(*

## Short summary
An interface to provide a scope selector for configurations in cycle managers.

.. <legal notes>

legal notes
=================
| SPDX-FileCopyrightText: © 2024 ekvip automation GmbH <info@ekvip.de>
| SPDX-License-Identifier: Apache-2.0
| For details check: Apache-2.0_

.. _Apache-2.0: https://www.apache.org/licenses/LICENSE-2.0

.. </legal notes>



*)
INTERFACE ICycleManagerConfigurationScope EXTENDS __SYSTEM.IQueryInterface

PROPERTY sequence : ISequenceConfiguration
GET
END_GET
END_PROPERTY

PROPERTY step : IStepConfiguration
GET
END_GET
END_PROPERTY

END_INTERFACE

(* stored: Version 1.1.0.1
   Itf ICycleManagerConfigurationScope: Id {c122f52e-d3a1-4c60-a305-86516c0d5d69}
   Property sequence: Id {d0fab6ee-0931-4bbf-97f7-0a8f613aeb45}
   Get Get: Id {76d3e71e-6c42-4f08-8095-6f219f39e954}
   Property step: Id {6b1a3255-99c7-49dc-9820-9c51898dbdb4}
   Get Get: Id {9d4fcf23-5044-45a6-9320-50626c390f52} *)
